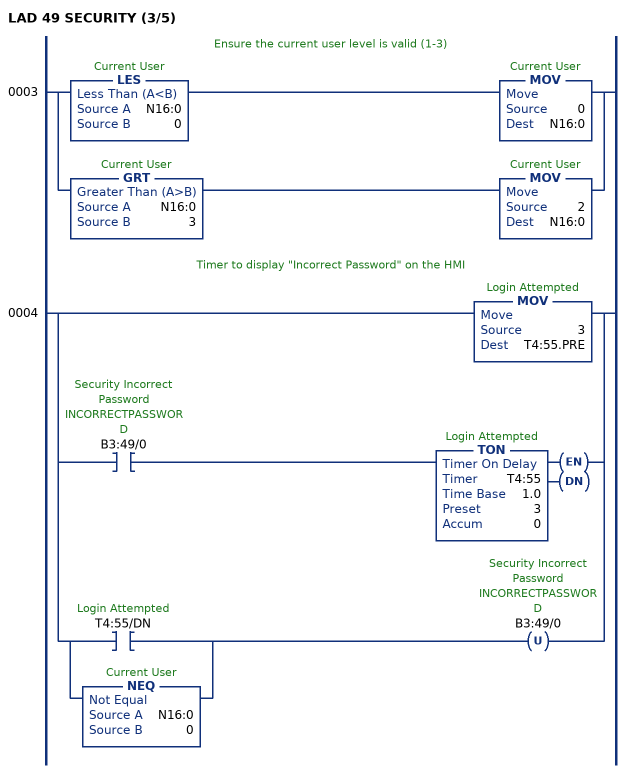
% Rung: 3 %
% Ensure the current user level is valid (1-3) %
SOR BST LES N16:0 0 MOV 0 N16:0 NXB GRT N16:0 3 MOV 2 N16:0 BND EOR
%   N16:0  "Current User" %
% Rung: 4 %
% Timer to display "Incorrect Password" on the HMI %
SOR BST MOV 3 T4:55.PRE NXB XIC B3:49/0 TON T4:55 1.0 3 0 NXB BST XIC T4:55/DN NXB NEQ N16:0 0 BND OTU B3:49/0 BND EOR
%   T4:55  "Login Attempted" %
%   B3:49/0  INCORRECTPASSWORD  "Security Incorrect Password" %
%   N16:0  "Current User" %

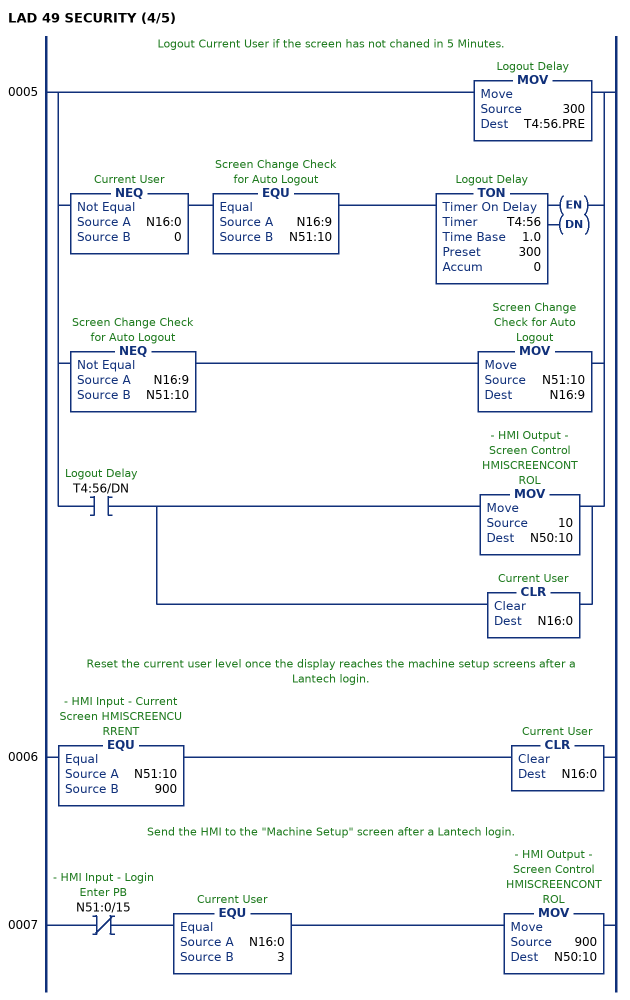
% Rung: 5 %
% Logout Current User if the screen has not chaned in 5 Minutes. %
SOR BST MOV 300 T4:56.PRE NXB NEQ N16:0 0 EQU N16:9 N51:10 TON T4:56 1.0 300 0 NXB NEQ N16:9 N51:10 MOV N51:10 N16:9 NXB XIC T4:56/DN BST MOV 10 N50:10 NXB CLR N16:0 BND BND EOR
%   T4:56  "Logout Delay" %
%   N16:0  "Current User" %
%   N16:9  "Screen Change Check for Auto Logout" %
%   N51:10  HMISCREENCURRENT  "- HMI Input - Current Screen" %
%   N50:10  HMISCREENCONTROL  "- HMI Output - Screen Control" %
% Rung: 6 %
% Reset the current user level once the display reaches the machine setup screens after a Lantech login. %
SOR EQU N51:10 900 CLR N16:0 EOR
%   N51:10  HMISCREENCURRENT  "- HMI Input - Current Screen" %
%   N16:0  "Current User" %
% Rung: 7 %
% Send the HMI to the "Machine Setup" screen after a Lantech login. %
SOR XIO N51:0/15 EQU N16:0 3 MOV 900 N50:10 EOR
%   N51:0/15  "- HMI Input - Login Enter PB" %
%   N16:0  "Current User" %
%   N50:10  HMISCREENCONTROL  "- HMI Output - Screen Control" %

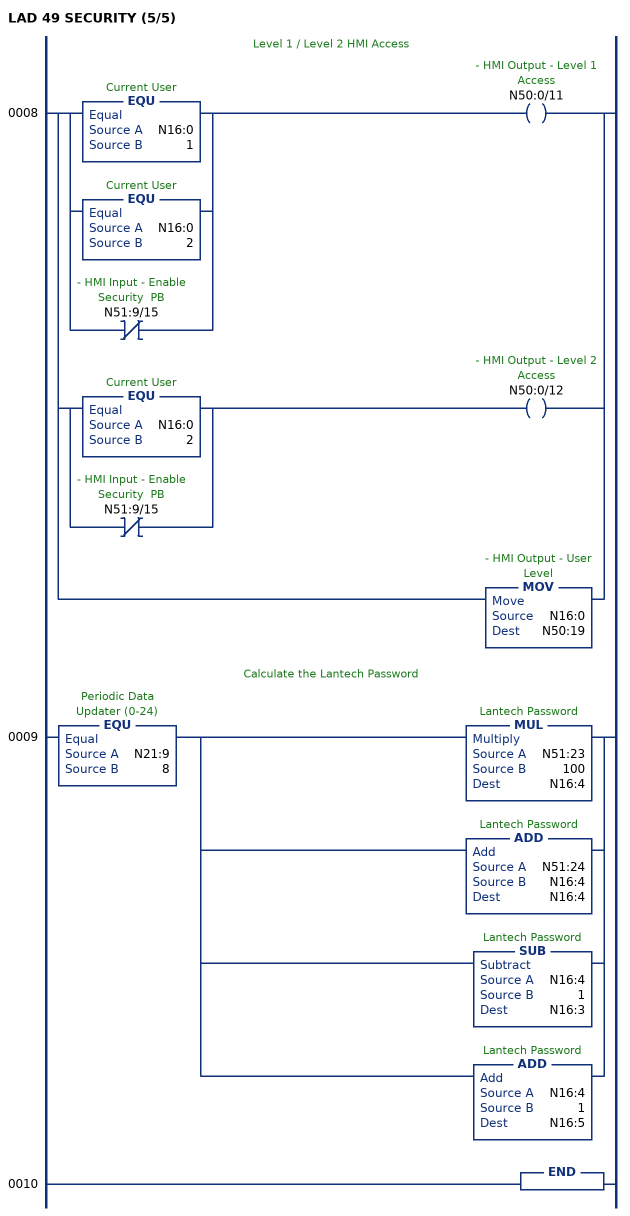
% Rung: 8 %
% Level 1 / Level 2 HMI Access %
SOR BST BST EQU N16:0 1 NXB EQU N16:0 2 NXB XIO N51:9/15 BND OTE N50:0/11 NXB BST EQU N16:0 2 NXB XIO N51:9/15 BND OTE N50:0/12 NXB MOV N16:0 N50:19 BND EOR
%   N16:0  "Current User" %
%   N51:9/15  "- HMI Input - Enable Security  PB" %
%   N50:0/11  "- HMI Output - Level 1 Access" %
%   N50:0/12  "- HMI Output - Level 2 Access" %
%   N50:19  "- HMI Output - User Level" %
% Rung: 9 %
% Calculate the Lantech Password %
SOR EQU N21:9 8 BST MUL N51:23 100 N16:4 NXB ADD N51:24 N16:4 N16:4 NXB SUB N16:4 1 N16:3 NXB ADD N16:4 1 N16:5 BND EOR
%   N21:9  "Periodic Data Updater (0-24)" %
%   N51:23  "- HMI Input - Hour" %
%   N16:4  "Lantech Password" %
%   N51:24  "- HMI Input - Minute" %
%   N16:3  "Lantech Password" %
%   N16:5  "Lantech Password" %
% Rung: 10 %
SOR END EOR

LADDER 50 "HMI"
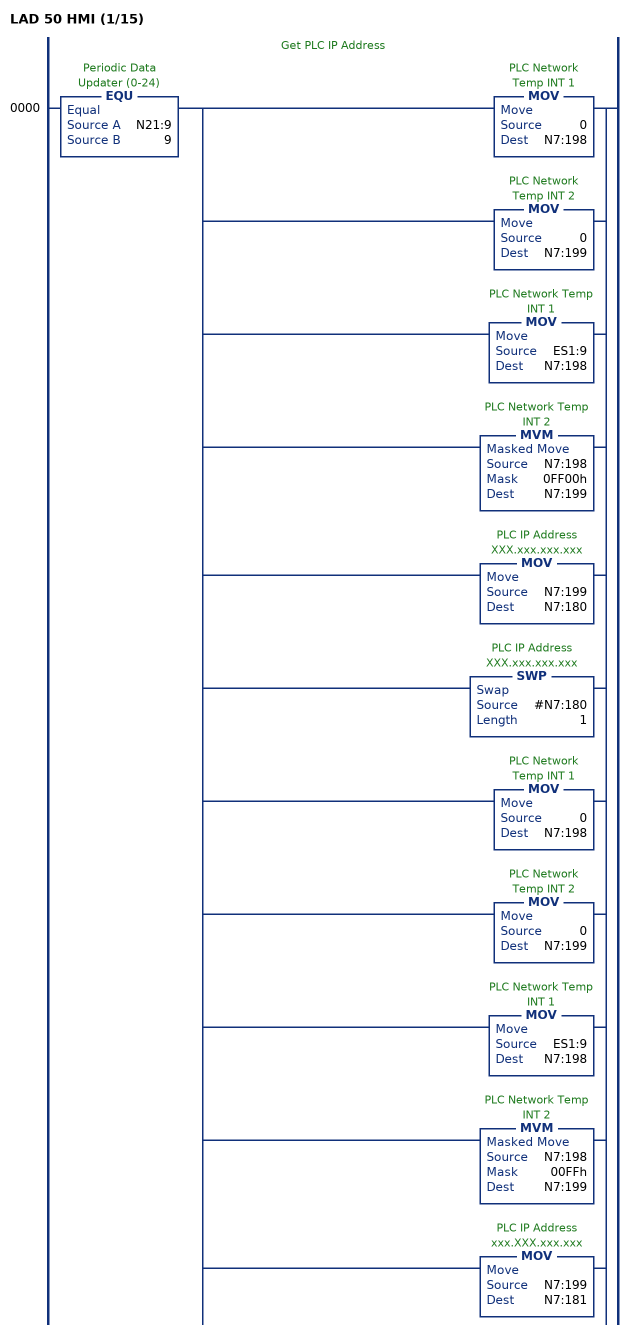
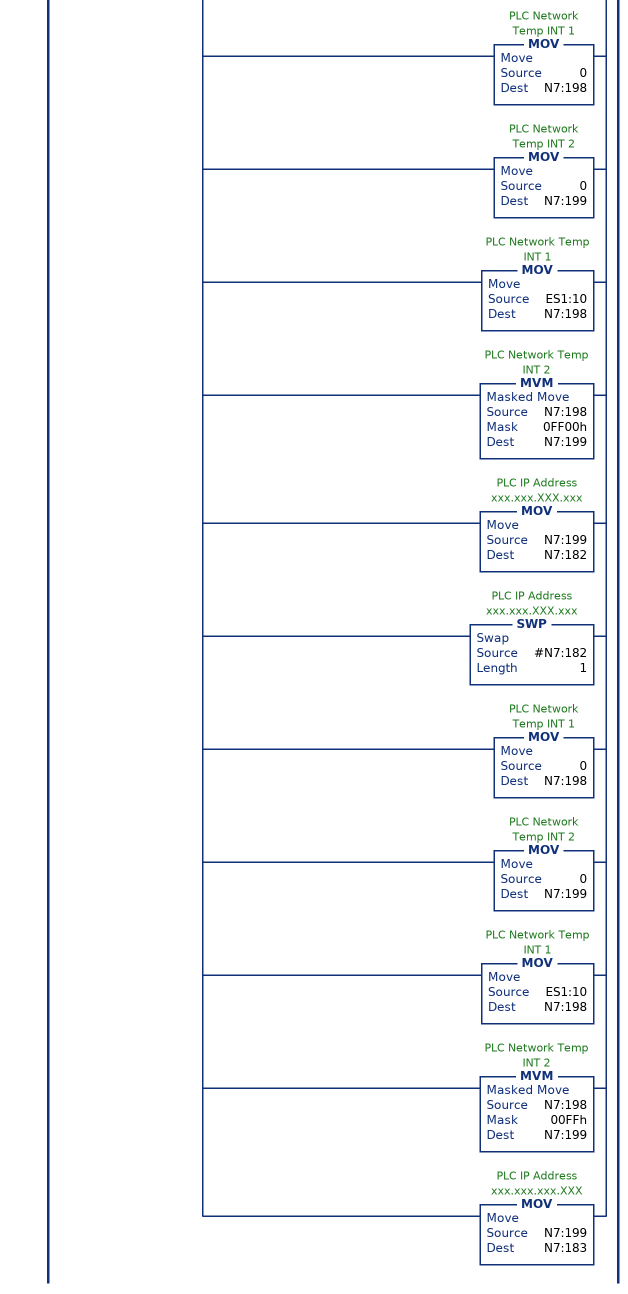
% Rung: 0 %
% Get PLC IP Address %
SOR EQU N21:9 9 BST BST MOV 0 N7:198 NXB MOV 0 N7:199 NXB MOV ES1:9 N7:198 NXB MVM N7:198 0FF00h N7:199 NXB MOV N7:199 N7:180 NXB SWP #N7:180 1 BND NXB BST MOV 0 N7:198 NXB MOV 0 N7:199 NXB MOV ES1:9 N7:198 NXB MVM N7:198 00FFh N7:199 NXB MOV N7:199 N7:181 BND NXB BST MOV 0 N7:198 NXB MOV 0 N7:199 NXB MOV ES1:10 N7:198 NXB MVM N7:198 0FF00h N7:199 NXB MOV N7:199 N7:182 NXB SWP #N7:182 1 BND NXB BST MOV 0 N7:198 NXB MOV 0 N7:199 NXB MOV ES1:10 N7:198 NXB MVM N7:198 00FFh N7:199 NXB MOV N7:199 N7:183 BND BND EOR
%   N21:9  "Periodic Data Updater (0-24)" %
%   N7:198  "PLC Network Temp INT 1" %
%   N7:199  "PLC Network Temp INT 2" %
%   N7:180  "PLC IP Address XXX.xxx.xxx.xxx" %
%   N7:181  "PLC IP Address xxx.XXX.xxx.xxx" %
%   N7:182  "PLC IP Address xxx.xxx.XXX.xxx" %
%   N7:183  "PLC IP Address xxx.xxx.xxx.XXX" %

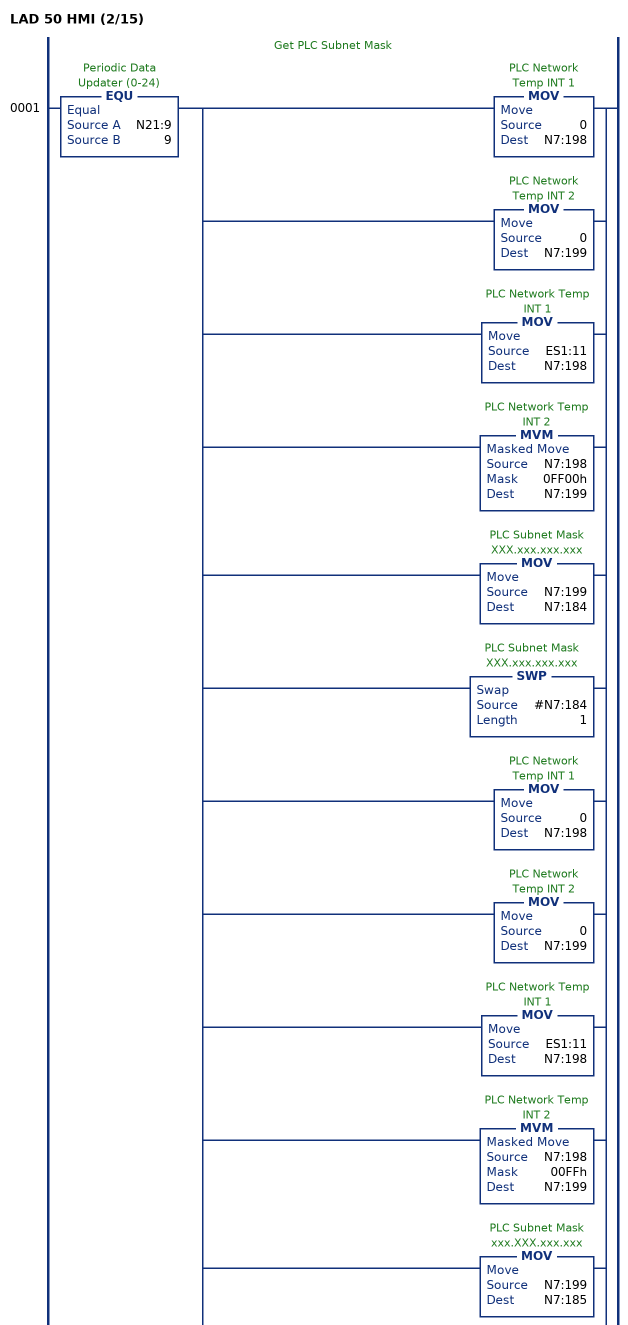

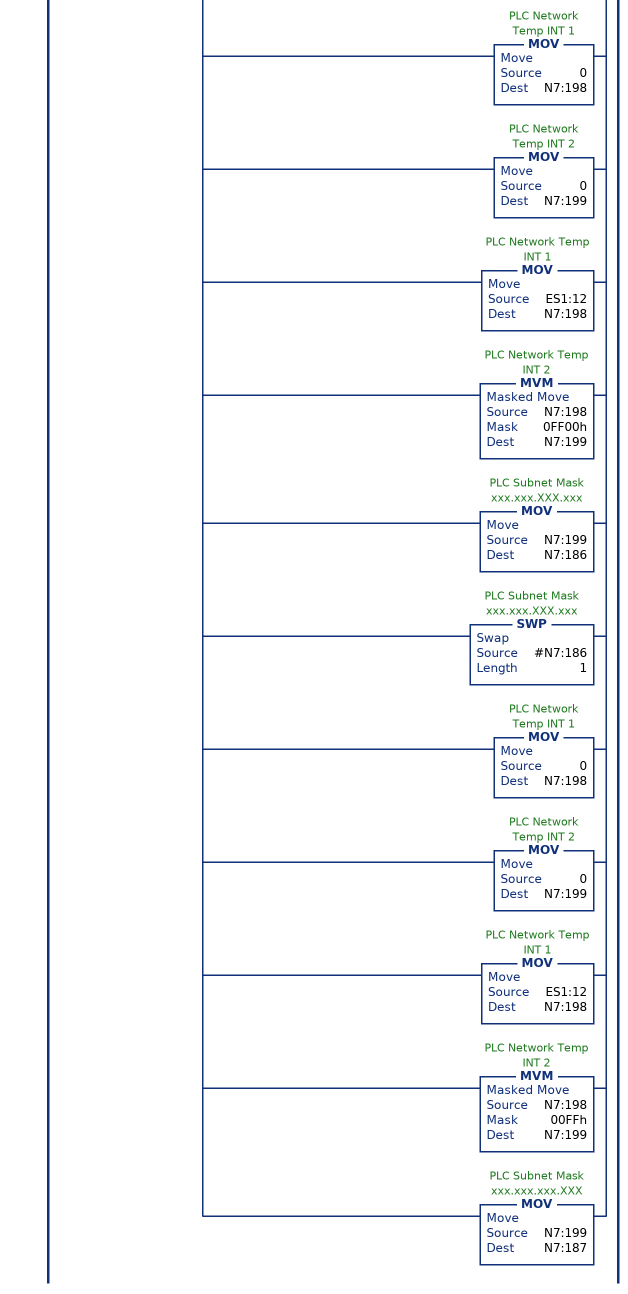
% Rung: 1 %
% Get PLC Subnet Mask %
SOR EQU N21:9 9 BST BST MOV 0 N7:198 NXB MOV 0 N7:199 NXB MOV ES1:11 N7:198 NXB MVM N7:198 0FF00h N7:199 NXB MOV N7:199 N7:184 NXB SWP #N7:184 1 BND NXB BST MOV 0 N7:198 NXB MOV 0 N7:199 NXB MOV ES1:11 N7:198 NXB MVM N7:198 00FFh N7:199 NXB MOV N7:199 N7:185 BND NXB BST MOV 0 N7:198 NXB MOV 0 N7:199 NXB MOV ES1:12 N7:198 NXB MVM N7:198 0FF00h N7:199 NXB MOV N7:199 N7:186 NXB SWP #N7:186 1 BND NXB BST MOV 0 N7:198 NXB MOV 0 N7:199 NXB MOV ES1:12 N7:198 NXB MVM N7:198 00FFh N7:199 NXB MOV N7:199 N7:187 BND BND EOR
%   N21:9  "Periodic Data Updater (0-24)" %
%   N7:198  "PLC Network Temp INT 1" %
%   N7:199  "PLC Network Temp INT 2" %
%   N7:184  "PLC Subnet Mask XXX.xxx.xxx.xxx" %
%   N7:185  "PLC Subnet Mask xxx.XXX.xxx.xxx" %
%   N7:186  "PLC Subnet Mask xxx.xxx.XXX.xxx" %
%   N7:187  "PLC Subnet Mask xxx.xxx.xxx.XXX" %

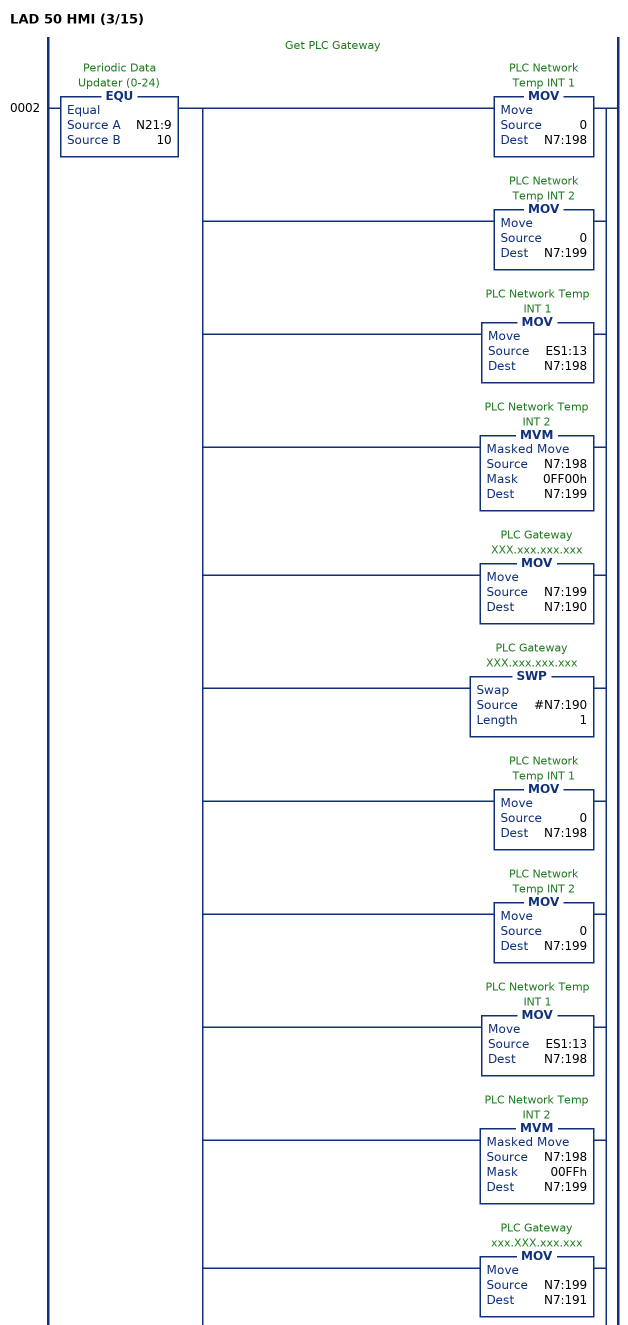

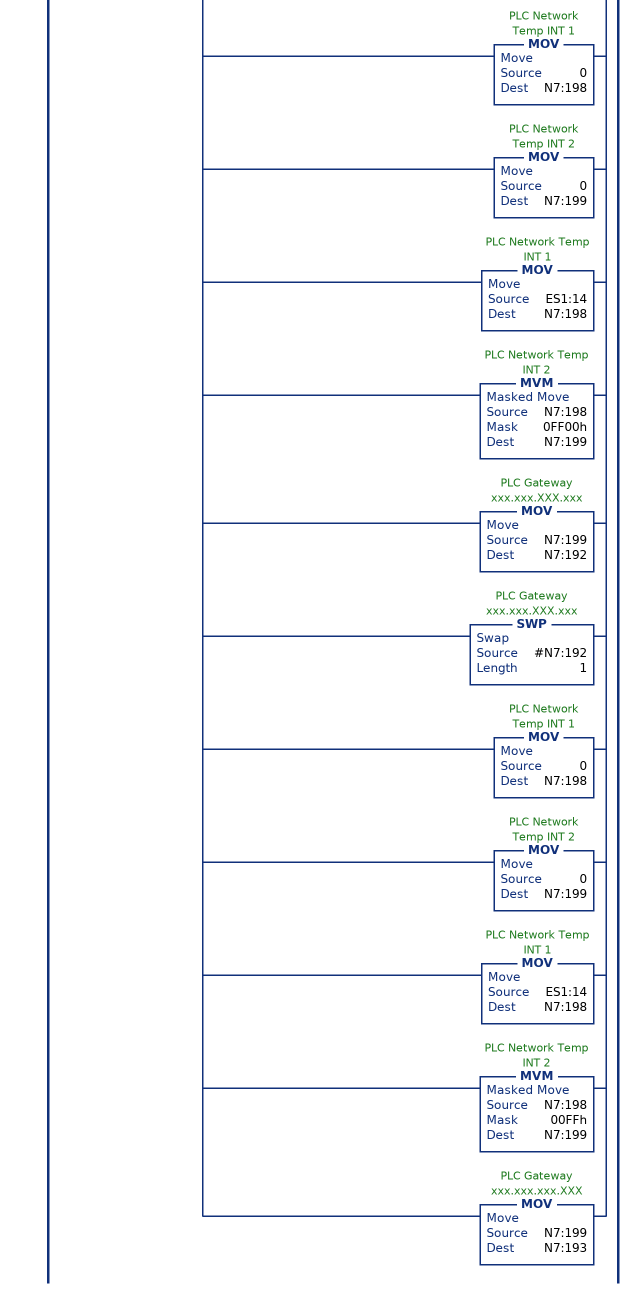
% Rung: 2 %
% Get PLC Gateway %
SOR EQU N21:9 10 BST BST MOV 0 N7:198 NXB MOV 0 N7:199 NXB MOV ES1:13 N7:198 NXB MVM N7:198 0FF00h N7:199 NXB MOV N7:199 N7:190 NXB SWP #N7:190 1 BND NXB BST MOV 0 N7:198 NXB MOV 0 N7:199 NXB MOV ES1:13 N7:198 NXB MVM N7:198 00FFh N7:199 NXB MOV N7:199 N7:191 BND NXB BST MOV 0 N7:198 NXB MOV 0 N7:199 NXB MOV ES1:14 N7:198 NXB MVM N7:198 0FF00h N7:199 NXB MOV N7:199 N7:192 NXB SWP #N7:192 1 BND NXB BST MOV 0 N7:198 NXB MOV 0 N7:199 NXB MOV ES1:14 N7:198 NXB MVM N7:198 00FFh N7:199 NXB MOV N7:199 N7:193 BND BND EOR
%   N21:9  "Periodic Data Updater (0-24)" %
%   N7:198  "PLC Network Temp INT 1" %
%   N7:199  "PLC Network Temp INT 2" %
%   N7:190  "PLC Gateway XXX.xxx.xxx.xxx" %
%   N7:191  "PLC Gateway xxx.XXX.xxx.xxx" %
%   N7:192  "PLC Gateway xxx.xxx.XXX.xxx" %
%   N7:193  "PLC Gateway xxx.xxx.xxx.XXX" %

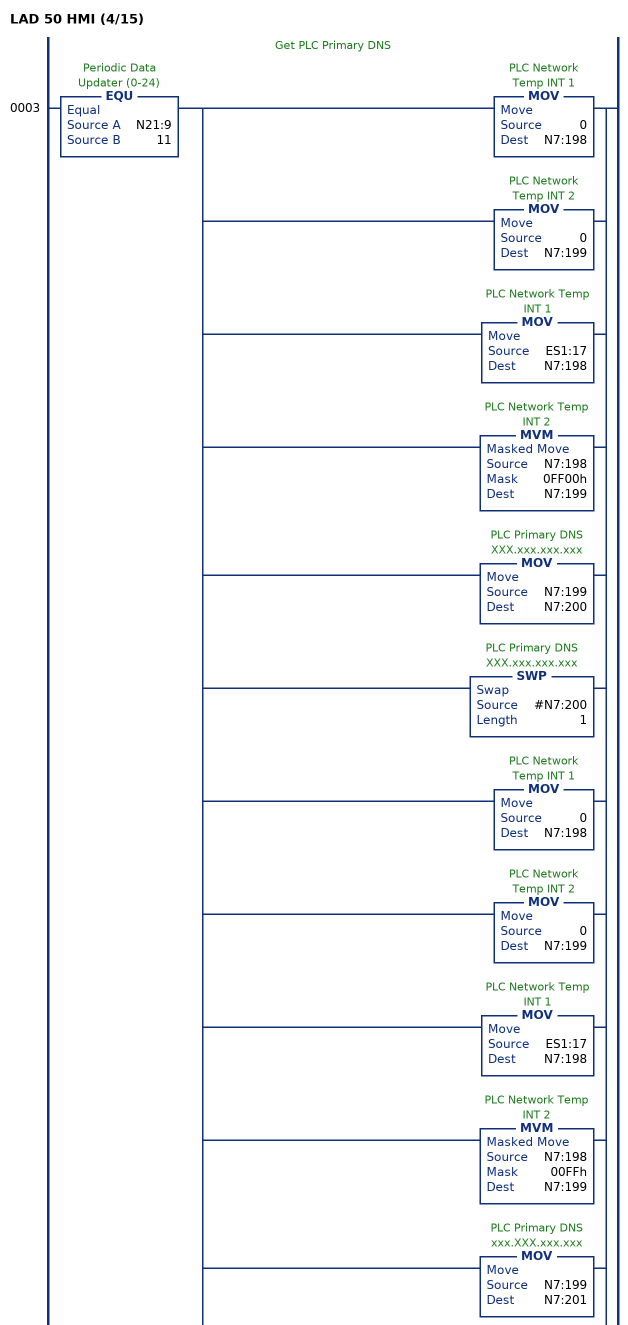

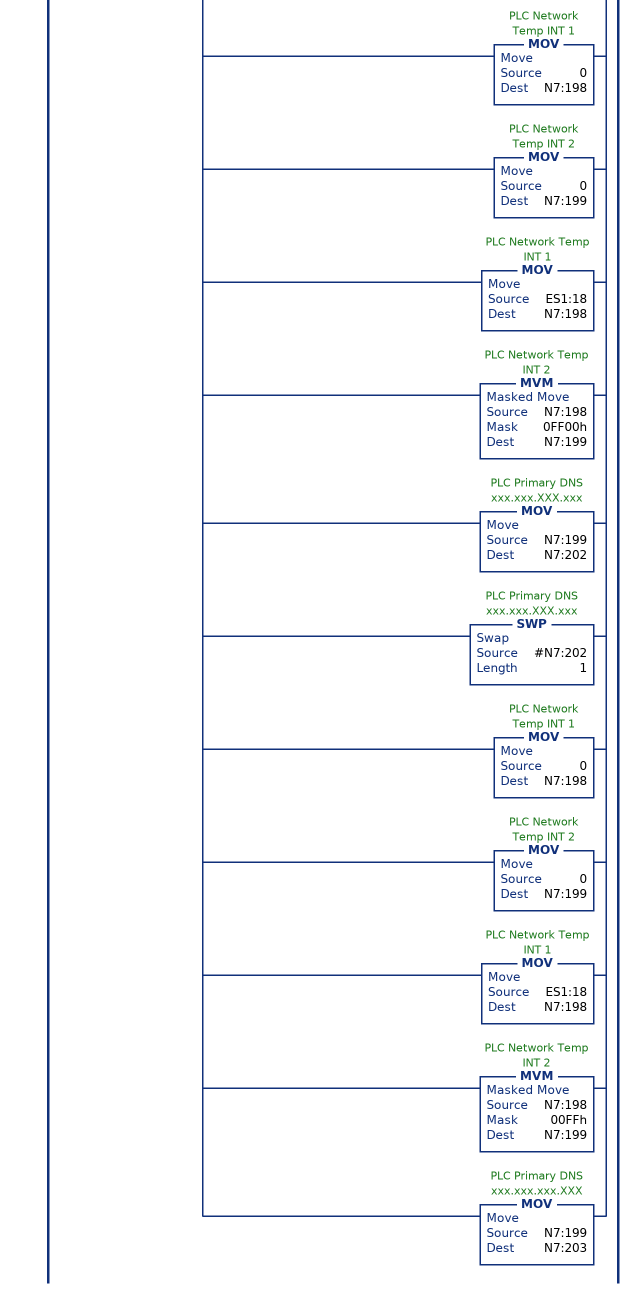
% Rung: 3 %
% Get PLC Primary DNS %
SOR EQU N21:9 11 BST BST MOV 0 N7:198 NXB MOV 0 N7:199 NXB MOV ES1:17 N7:198 NXB MVM N7:198 0FF00h N7:199 NXB MOV N7:199 N7:200 NXB SWP #N7:200 1 BND NXB BST MOV 0 N7:198 NXB MOV 0 N7:199 NXB MOV ES1:17 N7:198 NXB MVM N7:198 00FFh N7:199 NXB MOV N7:199 N7:201 BND NXB BST MOV 0 N7:198 NXB MOV 0 N7:199 NXB MOV ES1:18 N7:198 NXB MVM N7:198 0FF00h N7:199 NXB MOV N7:199 N7:202 NXB SWP #N7:202 1 BND NXB BST MOV 0 N7:198 NXB MOV 0 N7:199 NXB MOV ES1:18 N7:198 NXB MVM N7:198 00FFh N7:199 NXB MOV N7:199 N7:203 BND BND EOR
%   N21:9  "Periodic Data Updater (0-24)" %
%   N7:198  "PLC Network Temp INT 1" %
%   N7:199  "PLC Network Temp INT 2" %
%   N7:200  "PLC Primary DNS XXX.xxx.xxx.xxx" %
%   N7:201  "PLC Primary DNS xxx.XXX.xxx.xxx" %
%   N7:202  "PLC Primary DNS xxx.xxx.XXX.xxx" %
%   N7:203  "PLC Primary DNS xxx.xxx.xxx.XXX" %

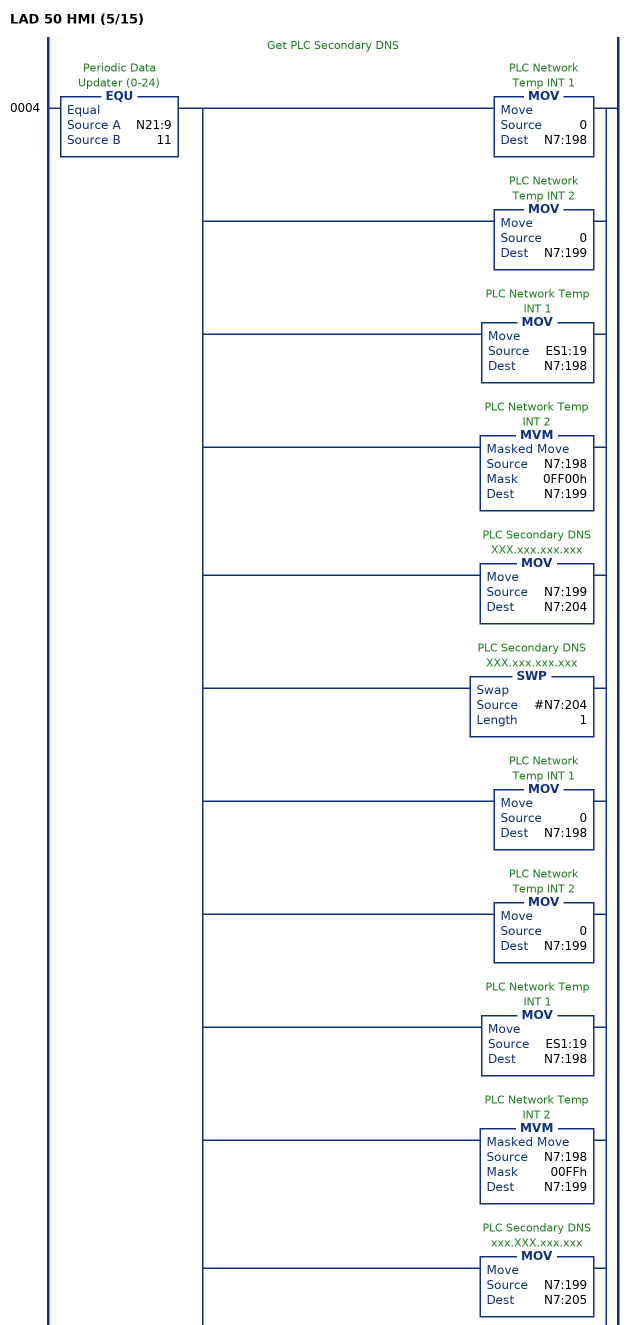

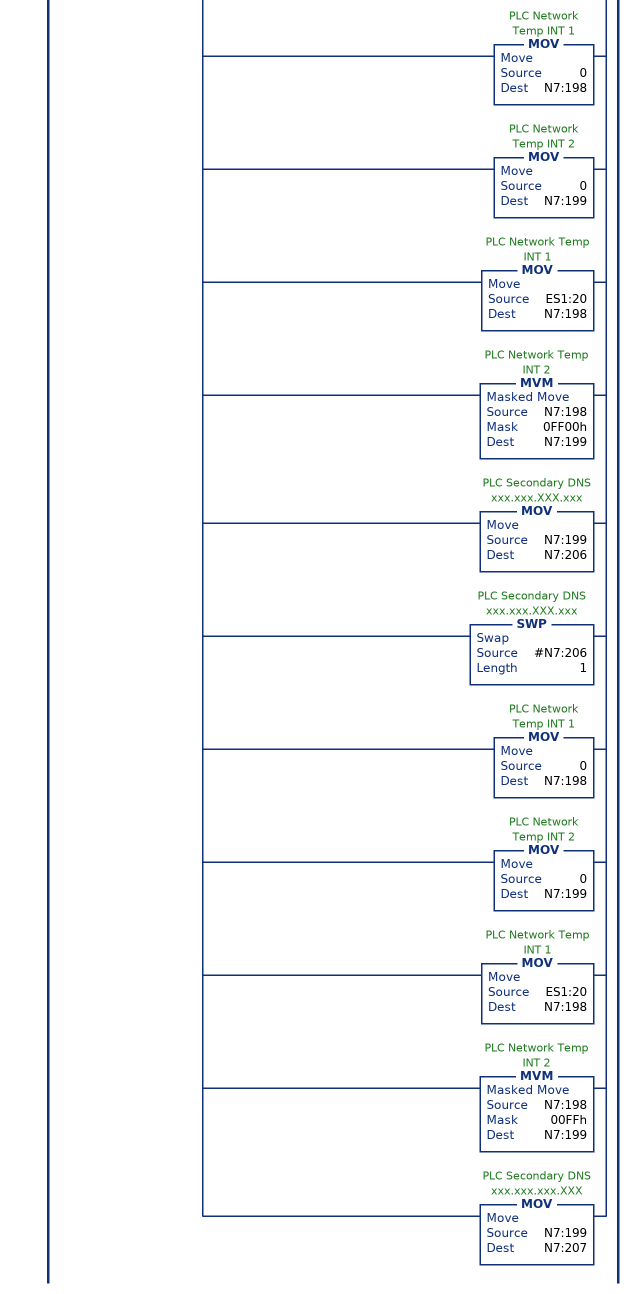
% Rung: 4 %
% Get PLC Secondary DNS %
SOR EQU N21:9 11 BST BST MOV 0 N7:198 NXB MOV 0 N7:199 NXB MOV ES1:19 N7:198 NXB MVM N7:198 0FF00h N7:199 NXB MOV N7:199 N7:204 NXB SWP #N7:204 1 BND NXB BST MOV 0 N7:198 NXB MOV 0 N7:199 NXB MOV ES1:19 N7:198 NXB MVM N7:198 00FFh N7:199 NXB MOV N7:199 N7:205 BND NXB BST MOV 0 N7:198 NXB MOV 0 N7:199 NXB MOV ES1:20 N7:198 NXB MVM N7:198 0FF00h N7:199 NXB MOV N7:199 N7:206 NXB SWP #N7:206 1 BND NXB BST MOV 0 N7:198 NXB MOV 0 N7:199 NXB MOV ES1:20 N7:198 NXB MVM N7:198 00FFh N7:199 NXB MOV N7:199 N7:207 BND BND EOR
%   N21:9  "Periodic Data Updater (0-24)" %
%   N7:198  "PLC Network Temp INT 1" %
%   N7:199  "PLC Network Temp INT 2" %
%   N7:204  "PLC Secondary DNS XXX.xxx.xxx.xxx" %
%   N7:205  "PLC Secondary DNS xxx.XXX.xxx.xxx" %
%   N7:206  "PLC Secondary DNS xxx.xxx.XXX.xxx" %
%   N7:207  "PLC Secondary DNS xxx.xxx.xxx.XXX" %

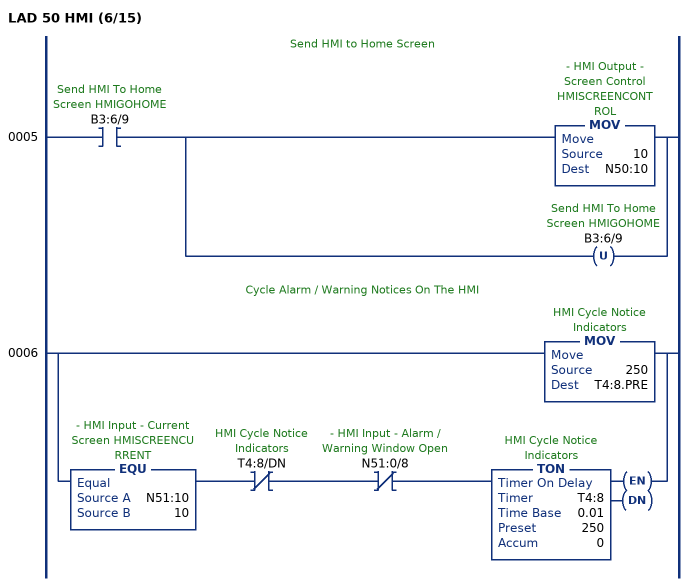
% Rung: 5 %
% Send HMI to Home Screen %
SOR XIC B3:6/9 BST MOV 10 N50:10 NXB OTU B3:6/9 BND EOR
%   B3:6/9  HMIGOHOME  "Send HMI To Home Screen" %
%   N50:10  HMISCREENCONTROL  "- HMI Output - Screen Control" %
% Rung: 6 %
% Cycle Alarm / Warning Notices On The HMI %
SOR BST MOV 250 T4:8.PRE NXB EQU N51:10 10 XIO T4:8/DN XIO N51:0/8 TON T4:8 0.01 250 0 BND EOR
%   T4:8  "HMI Cycle Notice Indicators" %
%   N51:10  HMISCREENCURRENT  "- HMI Input - Current Screen" %
%   N51:0/8  "- HMI Input - Alarm / Warning Window Open" %

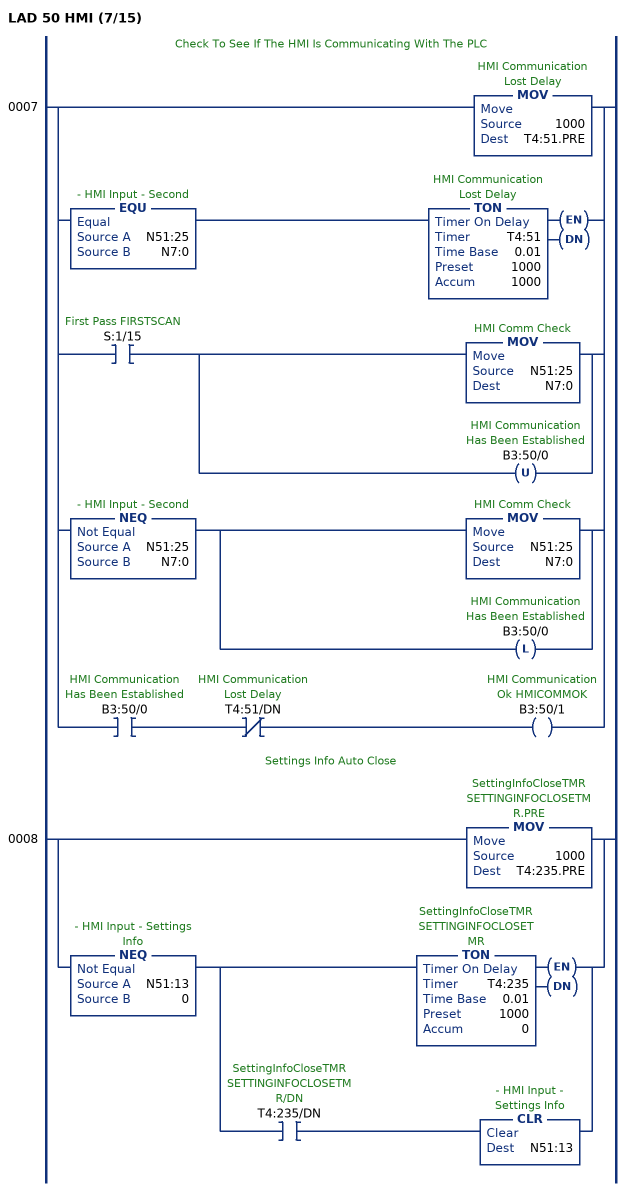
% Rung: 7 %
% Check To See If The HMI Is Communicating With The PLC %
SOR BST MOV 1000 T4:51.PRE NXB EQU N51:25 N7:0 TON T4:51 0.01 1000 1000 NXB XIC S:1/15 BST MOV N51:25 N7:0 NXB OTU B3:50/0 BND NXB NEQ N51:25 N7:0 BST MOV N51:25 N7:0 NXB OTL B3:50/0 BND NXB XIC B3:50/0 XIO T4:51/DN OTE B3:50/1 BND EOR
%   T4:51  "HMI Communication Lost Delay" %
%   N51:25  "- HMI Input - Second" %
%   N7:0  "HMI Comm Check" %
%   S:1/15  FIRSTSCAN  "First Pass" %
%   B3:50/0  "HMI Communication Has Been Established" %
%   B3:50/1  HMICOMMOK  "HMI Communication Ok" %
% Rung: 8 %
% Settings Info Auto Close %
SOR BST MOV 1000 T4:235.PRE NXB NEQ N51:13 0 BST TON T4:235 0.01 1000 0 NXB XIC T4:235/DN CLR N51:13 BND BND EOR
%   T4:235  SETTINGINFOCLOSETMR  "SettingInfoCloseTMR" %
%   N51:13  "- HMI Input - Settings Info" %

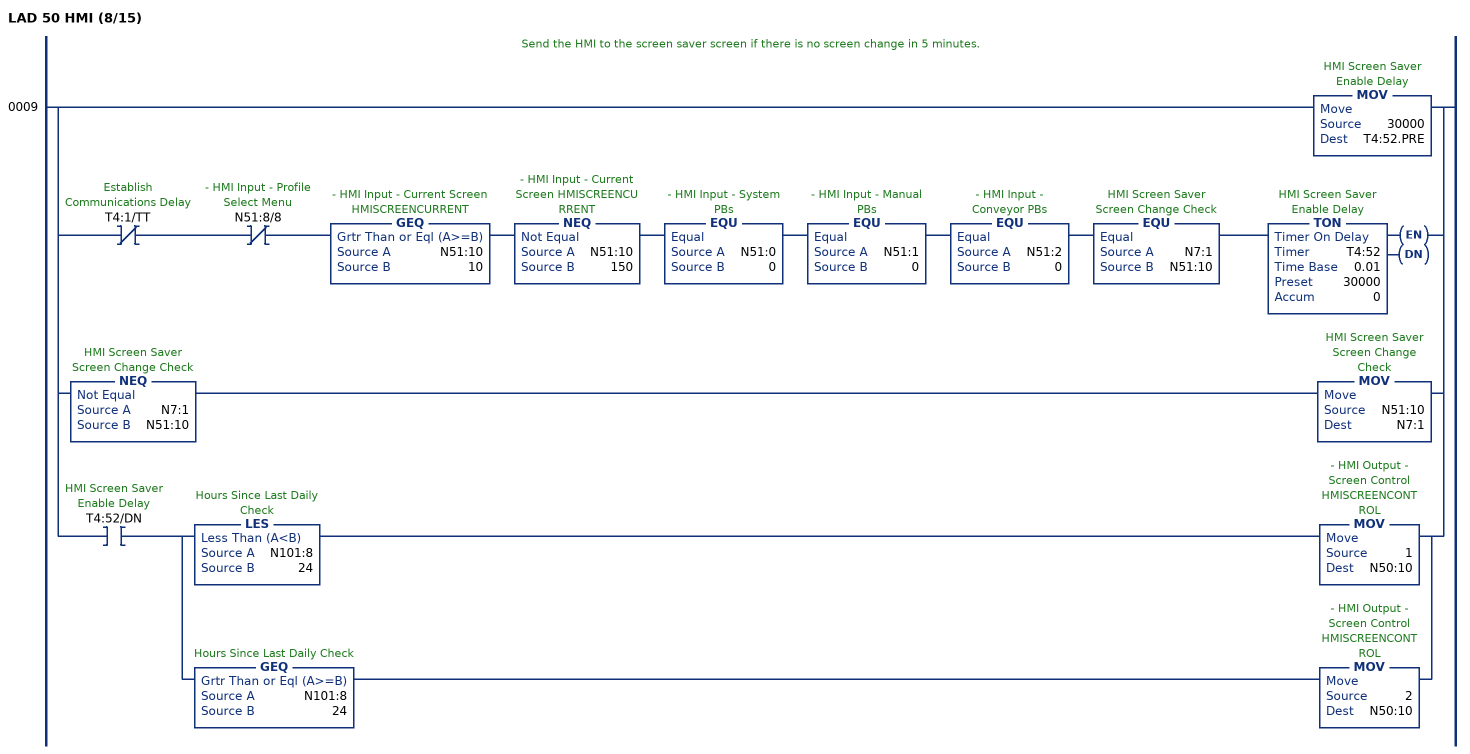
% Rung: 9 %
% Send the HMI to the screen saver screen if there is no screen change in 5 minutes. %
SOR BST MOV 30000 T4:52.PRE NXB XIO T4:1/TT XIO N51:8/8 GEQ N51:10 10 NEQ N51:10 150 EQU N51:0 0 EQU N51:1 0 EQU N51:2 0 EQU N7:1 N51:10 TON T4:52 0.01 30000 0 NXB NEQ N7:1 N51:10 MOV N51:10 N7:1 NXB XIC T4:52/DN BST LES N101:8 24 MOV 1 N50:10 NXB GEQ N101:8 24 MOV 2 N50:10 BND BND EOR
%   T4:52  "HMI Screen Saver Enable Delay" %
%   T4:1  "Establish Communications Delay" %
%   N51:8/8  "- HMI Input - Profile Select Menu" %
%   N51:10  HMISCREENCURRENT  "- HMI Input - Current Screen" %
%   N51:0  "- HMI Input - System PBs" %
%   N51:1  "- HMI Input - Manual PBs" %
%   N51:2  "- HMI Input - Conveyor PBs" %
%   N7:1  "HMI Screen Saver Screen Change Check" %
%   N101:8  "Hours Since Last Daily Check" %
%   N50:10  HMISCREENCONTROL  "- HMI Output - Screen Control" %

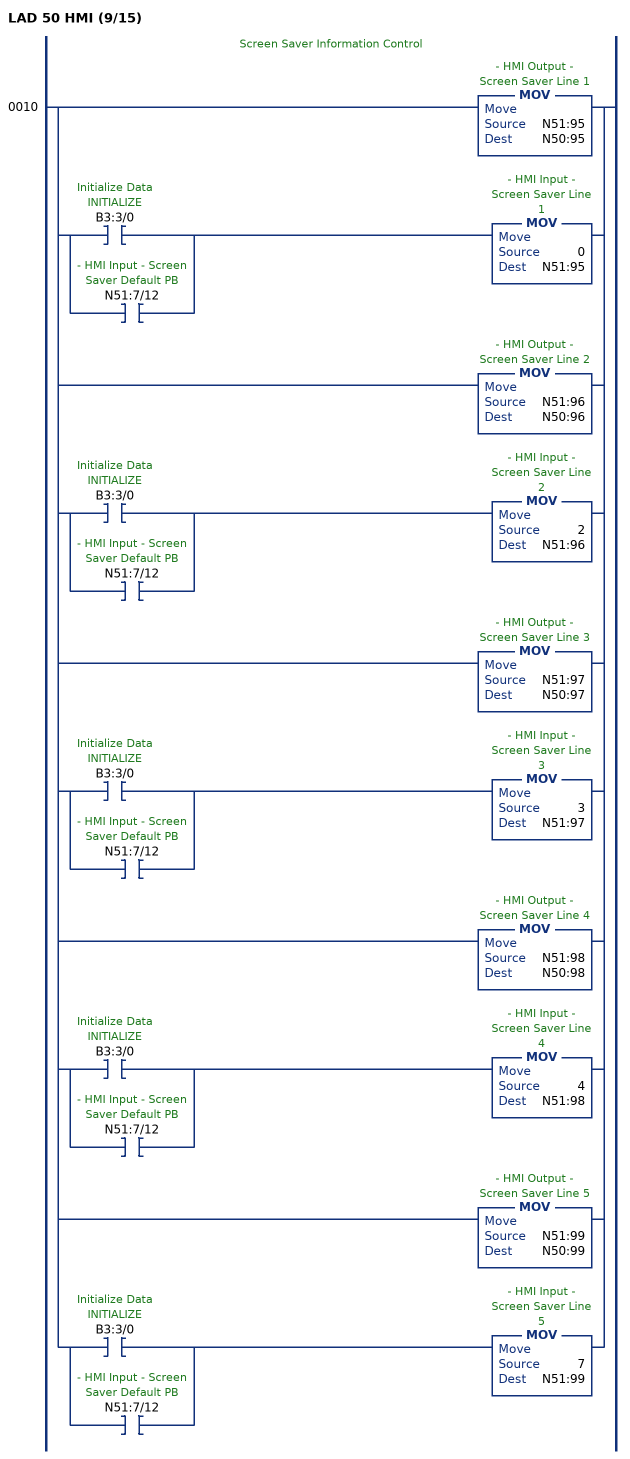
% Rung: 10 %
% Screen Saver Information Control %
SOR BST BST MOV N51:95 N50:95 NXB BST XIC B3:3/0 NXB XIC N51:7/12 BND MOV 0 N51:95 BND NXB BST MOV N51:96 N50:96 NXB BST XIC B3:3/0 NXB XIC N51:7/12 BND MOV 2 N51:96 BND NXB BST MOV N51:97 N50:97 NXB BST XIC B3:3/0 NXB XIC N51:7/12 BND MOV 3 N51:97 BND NXB BST MOV N51:98 N50:98 NXB BST XIC B3:3/0 NXB XIC N51:7/12 BND MOV 4 N51:98 BND NXB BST MOV N51:99 N50:99 NXB BST XIC B3:3/0 NXB XIC N51:7/12 BND MOV 7 N51:99 BND BND EOR
%   N51:95  "- HMI Input - Screen Saver Line 1" %
%   N50:95  "- HMI Output - Screen Saver Line 1" %
%   B3:3/0  INITIALIZE  "Initialize Data" %
%   N51:7/12  "- HMI Input - Screen Saver Default PB" %
%   N51:96  "- HMI Input - Screen Saver Line 2" %
%   N50:96  "- HMI Output - Screen Saver Line 2" %
%   N51:97  "- HMI Input - Screen Saver Line 3" %
%   N50:97  "- HMI Output - Screen Saver Line 3" %
%   N51:98  "- HMI Input - Screen Saver Line 4" %
%   N50:98  "- HMI Output - Screen Saver Line 4" %
%   N51:99  "- HMI Input - Screen Saver Line 5" %
%   N50:99  "- HMI Output - Screen Saver Line 5" %

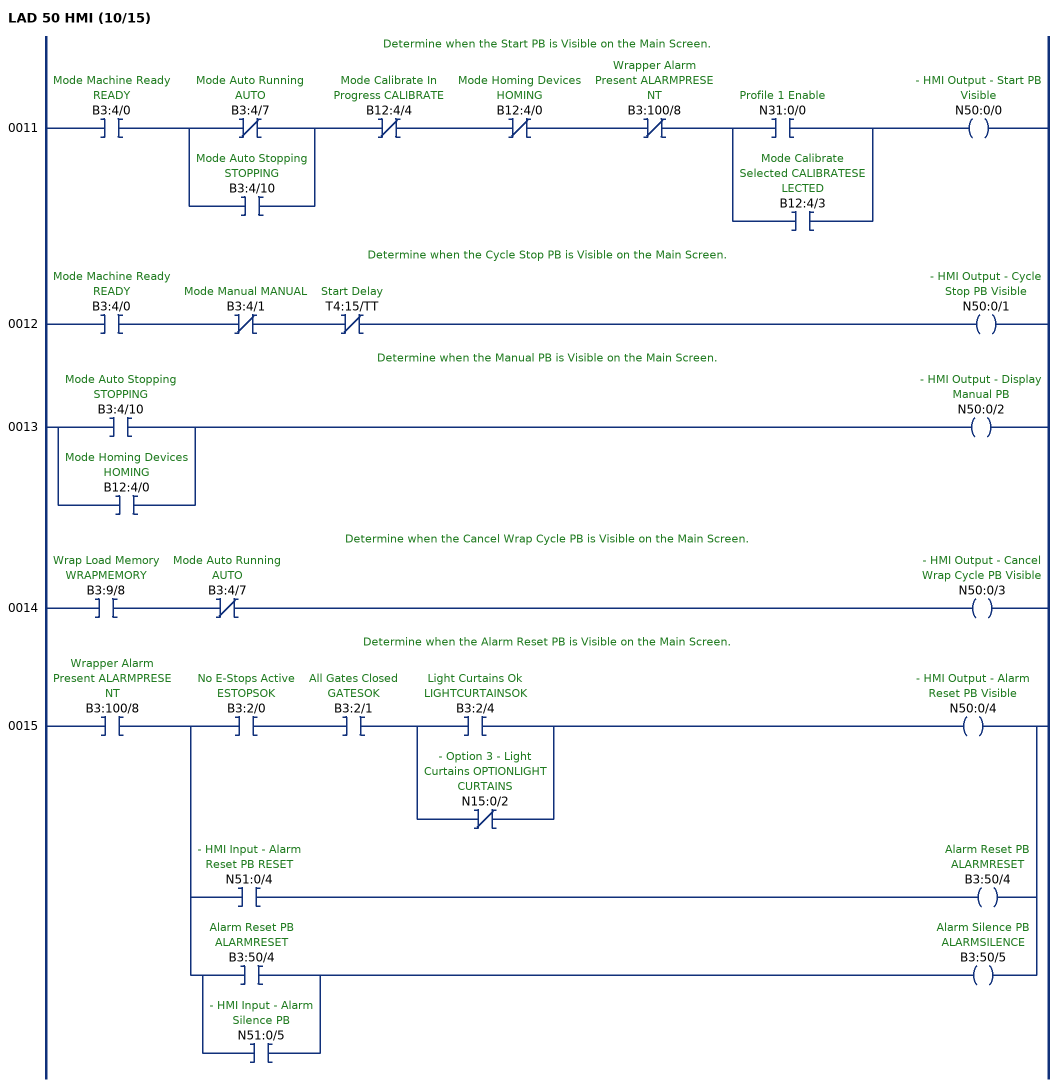
% Rung: 11 %
% Determine when the Start PB is Visible on the Main Screen. %
SOR XIC B3:4/0 BST XIO B3:4/7 NXB XIC B3:4/10 BND XIO B12:4/4 XIO B12:4/0 XIO B3:100/8 BST XIC N31:0/0 NXB XIC B12:4/3 BND OTE N50:0/0 EOR
%   B3:4/0  READY  "Mode Machine Ready" %
%   B3:4/7  AUTO  "Mode Auto Running" %
%   B3:4/10  STOPPING  "Mode Auto Stopping" %
%   B12:4/4  CALIBRATE  "Mode Calibrate In Progress" %
%   B12:4/0  HOMING  "Mode Homing Devices" %
%   B3:100/8  ALARMPRESENT  "Wrapper Alarm Present" %
%   N31:0/0  "Profile 1 Enable" %
%   B12:4/3  CALIBRATESELECTED  "Mode Calibrate Selected" %
%   N50:0/0  "- HMI Output - Start PB Visible" %
% Rung: 12 %
% Determine when the Cycle Stop PB is Visible on the Main Screen. %
SOR XIC B3:4/0 XIO B3:4/1 XIO T4:15/TT OTE N50:0/1 EOR
%   B3:4/0  READY  "Mode Machine Ready" %
%   B3:4/1  MANUAL  "Mode Manual" %
%   T4:15  "Start Delay" %
%   N50:0/1  "- HMI Output - Cycle Stop PB Visible" %
% Rung: 13 %
% Determine when the Manual PB is Visible on the Main Screen. %
SOR BST XIC B3:4/10 NXB XIC B12:4/0 BND OTE N50:0/2 EOR
%   B3:4/10  STOPPING  "Mode Auto Stopping" %
%   B12:4/0  HOMING  "Mode Homing Devices" %
%   N50:0/2  "- HMI Output - Display Manual PB" %
% Rung: 14 %
% Determine when the Cancel Wrap Cycle PB is Visible on the Main Screen. %
SOR XIC B3:9/8 XIO B3:4/7 OTE N50:0/3 EOR
%   B3:9/8  WRAPMEMORY  "Wrap Load Memory" %
%   B3:4/7  AUTO  "Mode Auto Running" %
%   N50:0/3  "- HMI Output - Cancel Wrap Cycle PB Visible" %
% Rung: 15 %
% Determine when the Alarm Reset PB is Visible on the Main Screen. %
SOR XIC B3:100/8 BST XIC B3:2/0 XIC B3:2/1 BST XIC B3:2/4 NXB XIO N15:0/2 BND OTE N50:0/4 NXB XIC N51:0/4 OTE B3:50/4 NXB BST XIC B3:50/4 NXB XIC N51:0/5 BND OTE B3:50/5 BND EOR
%   B3:100/8  ALARMPRESENT  "Wrapper Alarm Present" %
%   B3:2/0  ESTOPSOK  "No E-Stops Active" %
%   B3:2/1  GATESOK  "All Gates Closed" %
%   B3:2/4  LIGHTCURTAINSOK  "Light Curtains Ok" %
%   N15:0/2  OPTIONLIGHTCURTAINS  "- Option 3 - Light Curtains" %
%   N50:0/4  "- HMI Output - Alarm Reset PB Visible" %
%   N51:0/4  RESET  "- HMI Input - Alarm Reset PB" %
%   B3:50/4  ALARMRESET  "Alarm Reset PB" %
%   N51:0/5  "- HMI Input - Alarm Silence PB" %
%   B3:50/5  ALARMSILENCE  "Alarm Silence PB" %

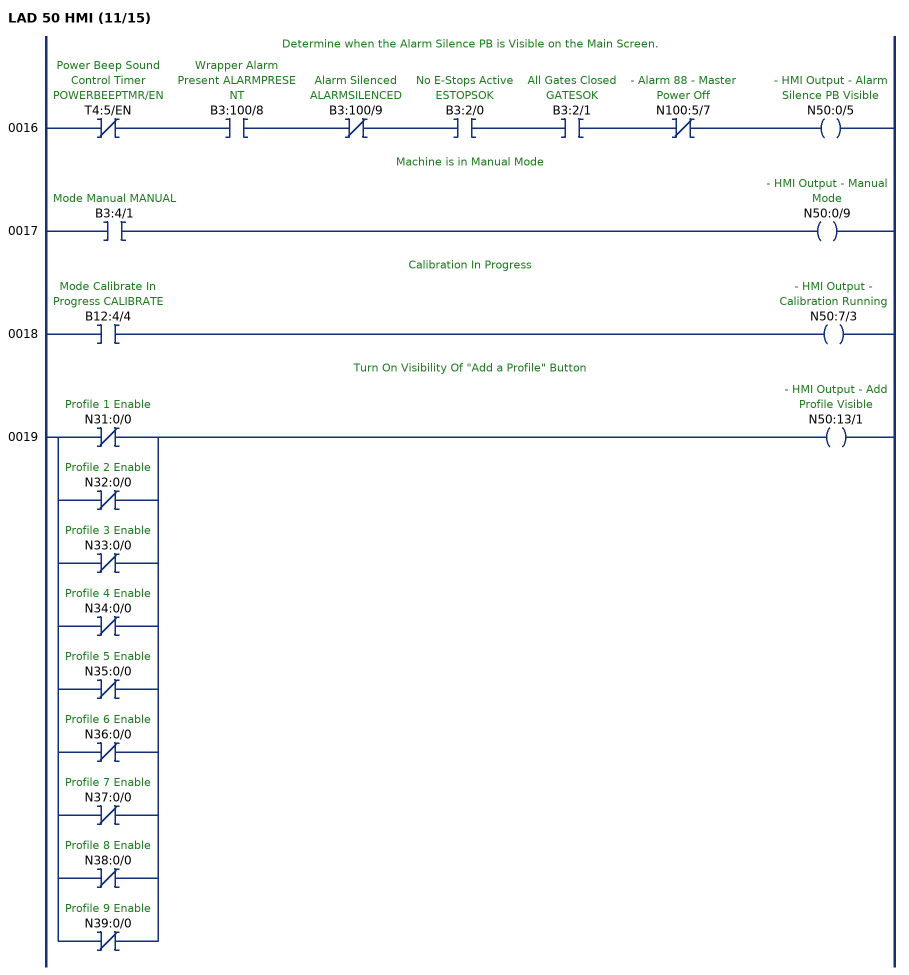
% Rung: 16 %
% Determine when the Alarm Silence PB is Visible on the Main Screen. %
SOR XIO T4:5/EN XIC B3:100/8 XIO B3:100/9 XIC B3:2/0 XIC B3:2/1 XIO N100:5/7 OTE N50:0/5 EOR
%   T4:5  POWERBEEPTMR  "Power Beep Sound Control Timer" %
%   B3:100/8  ALARMPRESENT  "Wrapper Alarm Present" %
%   B3:100/9  ALARMSILENCED  "Alarm Silenced" %
%   B3:2/0  ESTOPSOK  "No E-Stops Active" %
%   B3:2/1  GATESOK  "All Gates Closed" %
%   N100:5/7  "- Alarm 88 - Master Power Off" %
%   N50:0/5  "- HMI Output - Alarm Silence PB Visible" %
% Rung: 17 %
% Machine is in Manual Mode %
SOR XIC B3:4/1 OTE N50:0/9 EOR
%   B3:4/1  MANUAL  "Mode Manual" %
%   N50:0/9  "- HMI Output - Manual Mode" %
% Rung: 18 %
% Calibration In Progress %
SOR XIC B12:4/4 OTE N50:7/3 EOR
%   B12:4/4  CALIBRATE  "Mode Calibrate In Progress" %
%   N50:7/3  "- HMI Output - Calibration Running" %
% Rung: 19 %
% Turn On Visibility Of "Add a Profile" Button %
SOR BST XIO N31:0/0 NXB XIO N32:0/0 NXB XIO N33:0/0 NXB XIO N34:0/0 NXB XIO N35:0/0 NXB XIO N36:0/0 NXB XIO N37:0/0 NXB XIO N38:0/0 NXB XIO N39:0/0 BND OTE N50:13/1 EOR
%   N31:0/0  "Profile 1 Enable" %
%   N32:0/0  "Profile 2 Enable" %
%   N33:0/0  "Profile 3 Enable" %
%   N34:0/0  "Profile 4 Enable" %
%   N35:0/0  "Profile 5 Enable" %
%   N36:0/0  "Profile 6 Enable" %
%   N37:0/0  "Profile 7 Enable" %
%   N38:0/0  "Profile 8 Enable" %
%   N39:0/0  "Profile 9 Enable" %
%   N50:13/1  "- HMI Output - Add Profile Visible" %

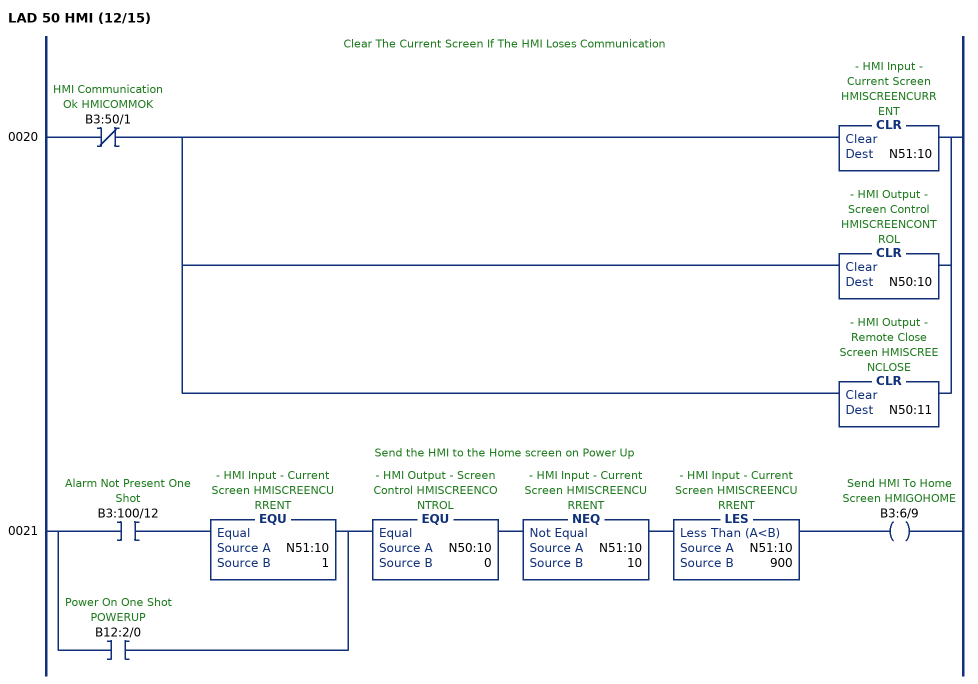
% Rung: 20 %
% Clear The Current Screen If The HMI Loses Communication %
SOR XIO B3:50/1 BST CLR N51:10 NXB CLR N50:10 NXB CLR N50:11 BND EOR
%   B3:50/1  HMICOMMOK  "HMI Communication Ok" %
%   N51:10  HMISCREENCURRENT  "- HMI Input - Current Screen" %
%   N50:10  HMISCREENCONTROL  "- HMI Output - Screen Control" %
%   N50:11  HMISCREENCLOSE  "- HMI Output - Remote Close Screen" %
% Rung: 21 %
% Send the HMI to the Home screen on Power Up %
SOR BST XIC B3:100/12 EQU N51:10 1 NXB XIC B12:2/0 BND EQU N50:10 0 NEQ N51:10 10 LES N51:10 900 OTE B3:6/9 EOR
%   B3:100/12  "Alarm Not Present One Shot" %
%   N51:10  HMISCREENCURRENT  "- HMI Input - Current Screen" %
%   B12:2/0  POWERUP  "Power On One Shot" %
%   N50:10  HMISCREENCONTROL  "- HMI Output - Screen Control" %
%   B3:6/9  HMIGOHOME  "Send HMI To Home Screen" %

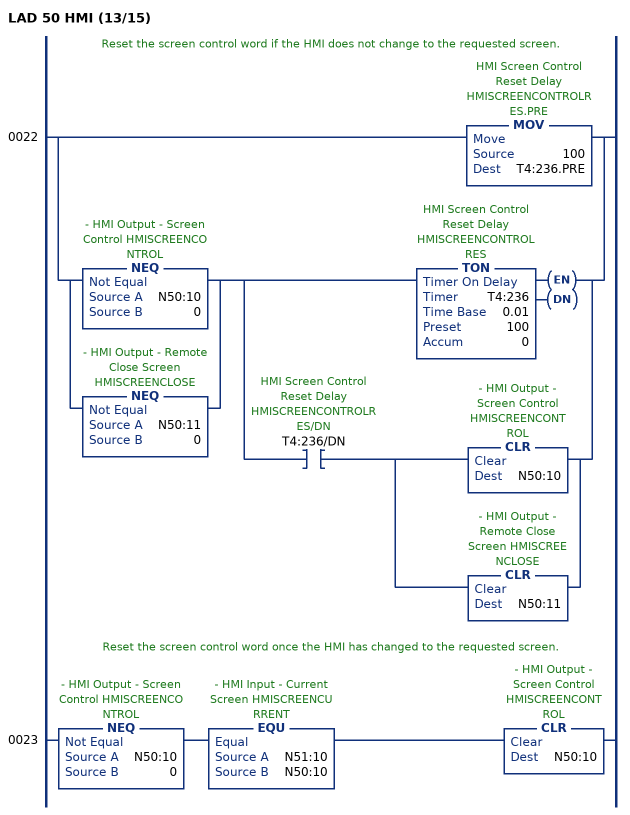
% Rung: 22 %
% Reset the screen control word if the HMI does not change to the requested screen. %
SOR BST MOV 100 T4:236.PRE NXB BST NEQ N50:10 0 NXB NEQ N50:11 0 BND BST TON T4:236 0.01 100 0 NXB XIC T4:236/DN BST CLR N50:10 NXB CLR N50:11 BND BND BND EOR
%   T4:236  HMISCREENCONTROLRES  "HMI Screen Control Reset Delay" %
%   N50:10  HMISCREENCONTROL  "- HMI Output - Screen Control" %
%   N50:11  HMISCREENCLOSE  "- HMI Output - Remote Close Screen" %
% Rung: 23 %
% Reset the screen control word once the HMI has changed to the requested screen. %
SOR NEQ N50:10 0 EQU N51:10 N50:10 CLR N50:10 EOR
%   N50:10  HMISCREENCONTROL  "- HMI Output - Screen Control" %
%   N51:10  HMISCREENCURRENT  "- HMI Input - Current Screen" %

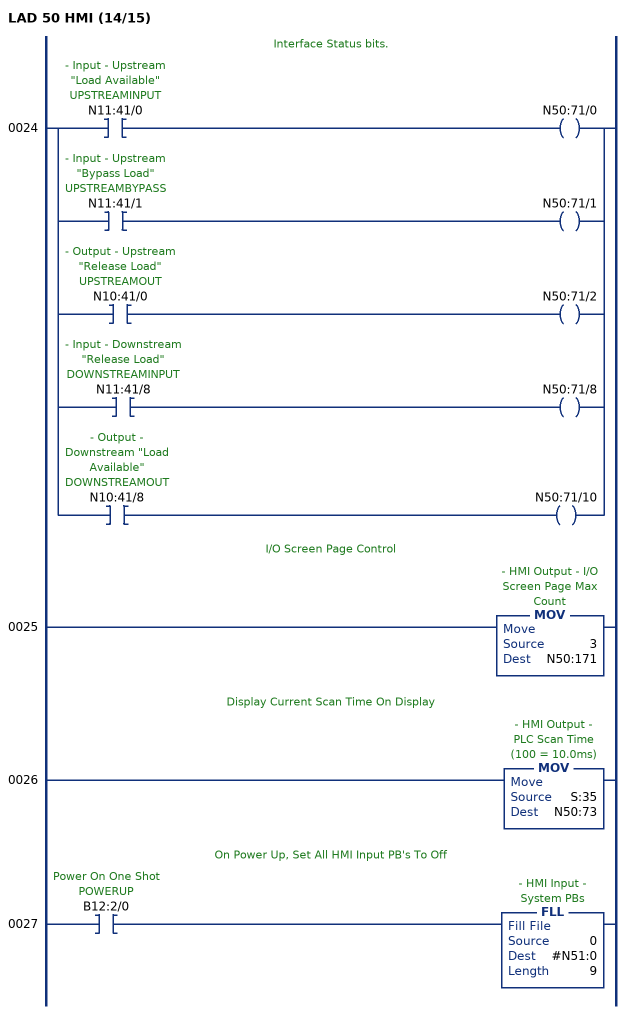
% Rung: 24 %
% Interface Status bits. %
SOR BST XIC N11:41/0 OTE N50:71/0 NXB XIC N11:41/1 OTE N50:71/1 NXB XIC N10:41/0 OTE N50:71/2 NXB XIC N11:41/8 OTE N50:71/8 NXB XIC N10:41/8 OTE N50:71/10 BND EOR
%   N11:41/0  UPSTREAMINPUT  "- Input - Upstream "Load Available"" %
%   N11:41/1  UPSTREAMBYPASS  "- Input - Upstream "Bypass Load"" %
%   N10:41/0  UPSTREAMOUT  "- Output - Upstream "Release Load"" %
%   N11:41/8  DOWNSTREAMINPUT  "- Input - Downstream "Release Load"" %
%   N10:41/8  DOWNSTREAMOUT  "- Output - Downstream "Load Available"" %
% Rung: 25 %
% I/O Screen Page Control %
SOR MOV 3 N50:171 EOR
%   N50:171  "- HMI Output - I/O Screen Page Max Count" %
% Rung: 26 %
% Display Current Scan Time On Display %
SOR MOV S:35 N50:73 EOR
%   S:35  "Last 1 ms Scan Time" %
%   N50:73  "- HMI Output - PLC Scan Time (100 = 10.0ms)" %
% Rung: 27 %
% On Power Up, Set All HMI Input PB's To Off %
SOR XIC B12:2/0 FLL 0 #N51:0 9 EOR
%   B12:2/0  POWERUP  "Power On One Shot" %
%   N51:0  "- HMI Input - System PBs" %

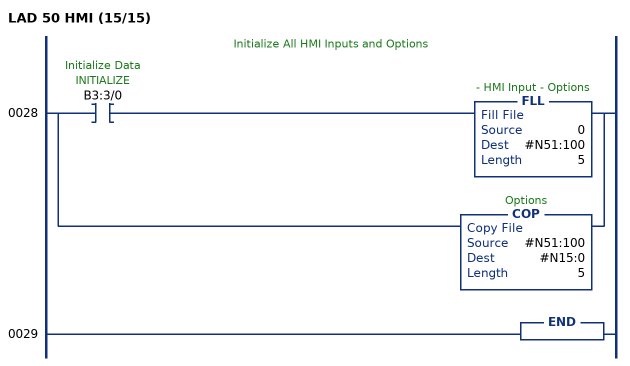
% Rung: 28 %
% Initialize All HMI Inputs and Options %
SOR BST XIC B3:3/0 FLL 0 #N51:100 5 NXB COP #N51:100 #N15:0 5 BND EOR
%   B3:3/0  INITIALIZE  "Initialize Data" %
%   N51:100  "- HMI Input - Options" %
%   N15:0  "Options" %
% Rung: 29 %
SOR END EOR

LADDER 52 "CYCLE INFO"
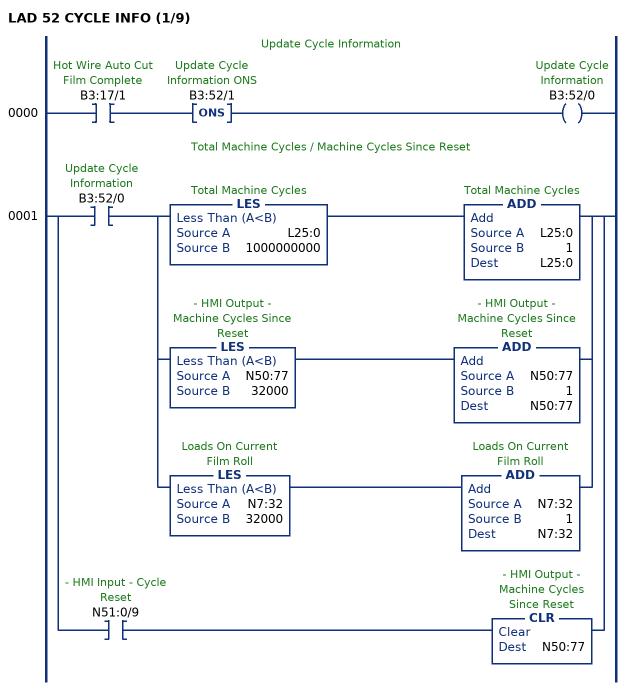
% Rung: 0 %
% Update Cycle Information %
SOR XIC B3:17/1 ONS B3:52/1 OTE B3:52/0 EOR
%   B3:17/1  "Hot Wire Auto Cut Film Complete" %
%   B3:52/1  "Update Cycle Information ONS" %
%   B3:52/0  "Update Cycle Information" %
% Rung: 1 %
% Total Machine Cycles / Machine Cycles Since Reset %
SOR BST XIC B3:52/0 BST LES L25:0 1000000000 ADD L25:0 1 L25:0 NXB LES N50:77 32000 ADD N50:77 1 N50:77 NXB LES N7:32 32000 ADD N7:32 1 N7:32 BND NXB XIC N51:0/9 CLR N50:77 BND EOR
%   B3:52/0  "Update Cycle Information" %
%   L25:0  "Total Machine Cycles" %
%   N50:77  "- HMI Output - Machine Cycles Since Reset" %
%   N7:32  "Loads On Current Film Roll" %
%   N51:0/9  "- HMI Input - Cycle Reset" %

